# B&R Automation Studio project prak11
Automation Studio 4.5.2.102

## Configuration Config1

### Hardware
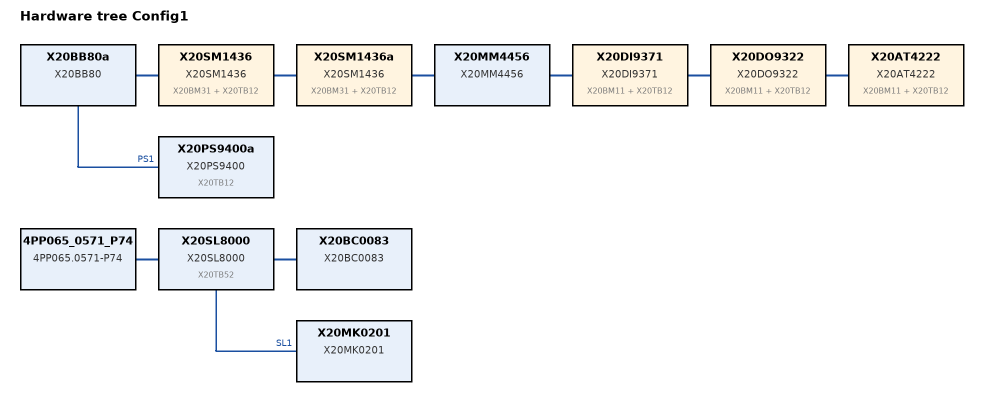
```
4PP065_0571_P74 : 4PP065.0571-P74 v1.1.2.0
  Connector IF5:
    ActivateDevice = 1
    Mode = Manual
    InternetAddress = 10.0.1.10
    SubnetMask = 255.255.255.0
  ConfigurationID = labBR
  TimerDeviceType = EPLX2X
  TimerDevice = 4PP065_0571_P74.IF4
  TaskClassIdleTime = 2000
  Cyclic1Output = 1
X20AT4222 : X20AT4222 v1.2.3.0  [SS1 -> X20TB12e.SS; SL -> X20BM11b.SL1]
X20BB80a : X20BB80 v1.0.2.0
X20BC0083 : X20BC0083 v2.9.0.0  [PLK1 -> X20SL8000.PLK2 [Cable Type=PowerlinkCable, Length=10, Version=1.0.0.2]; SL -> X20BB80a.SL1]
X20BM11 : X20BM11 v1.0.0.1  [X2X1 -> X20MM4456.X2X2]
X20BM11a : X20BM11 v1.0.0.1  [X2X1 -> X20BM11.X2X2]
X20BM11b : X20BM11 v1.0.0.1  [X2X1 -> X20BM11a.X2X2]
X20BM31 : X20BM31 v1.0.0.1  [X2X1 -> X20BB80a.IF1]
X20BM31a : X20BM31 v1.0.0.1  [X2X1 -> X20BM31.X2X2]
X20DI9371 : X20DI9371 v1.0.2.0  [SS1 -> X20TB12c.SS; SL -> X20BM11.SL1]
X20DO9322 : X20DO9322 v1.0.3.0  [SS1 -> X20TB12d.SS; SL -> X20BM11a.SL1]
X20MK0201 : X20MK0201 v1.0.0.0  [SL -> X20SL8000.SL1]
X20MM4456 : X20MM4456 v1.1.5.0  [X2X1 -> X20BM31a.X2X2]
X20PS9400a : X20PS9400 v1.0.2.4  [SS1 -> X20TB12a.SS; PS -> X20BB80a.PS1]
X20SL8000 : X20SL8000 v1.6.5.1  [PLK1 -> 4PP065_0571_P74.IF4 [Cable Type=PowerlinkCable, Length=10, Version=1.0.0.2]; PLK2 -> X20BC0083.PLK1 [Cable Type=PowerlinkCable, Length=10, Version=1.0.0.2]; SS1 -> X20TB52.SS]
  SafeProject = SafeLOGIC-1
X20SM1436 : X20SM1436 v1.4.2.1  [SS1 -> X20TB12.SS; SL -> X20BM31.SL1]
X20SM1436a : X20SM1436 v1.4.2.1  [SS1 -> X20TB12b.SS; SL -> X20BM31a.SL1]
X20TB12 : X20TB12 v1.0.0.0
X20TB12a : X20TB12 v1.0.0.0
X20TB12b : X20TB12 v1.0.0.0
X20TB12c : X20TB12 v1.0.0.0
X20TB12d : X20TB12 v1.0.0.0
X20TB12e : X20TB12 v1.0.0.0
X20TB52 : X20TB52 v1.0.0.1
```

## Logical view

### Global.var
```iecst
VAR
	led1 : {REDUND_UNREPLICABLE} BOOL;
	led2 : {REDUND_UNREPLICABLE} BOOL;
	led3 : {REDUND_UNREPLICABLE} BOOL;
	led4 : {REDUND_UNREPLICABLE} BOOL;
END_VAR
```

### Program Logical/Program

#### Main.c
```c
#include <bur/plctypes.h>

#ifdef _DEFAULT_INCLUDES
	#include <AsDefault.h>
#endif

void _INIT ProgramInit(void)
{
	i = 0;
}

void _CYCLIC ProgramCyclic(void)
{
	led1 = !led1;
	if(i%2)
	{
		led2 = !led2;
	}
	i++;
}

void _EXIT ProgramExit(void)
{

}
```
